{attribute 'pack_mode' := '1'}
TYPE ST_MqttMessage :
STRUCT
	sTopic : STRING;
	sMessage : T_MAXSTRING;
END_STRUCT
END_TYPE

(* stored: Version 1.1.0.1, ProductVersion 3.1.4024.2
   POU ST_MqttMessage: Id {89c0be22-c749-48c2-873e-ede4c6b89015}, SpecialFunc None *)
